// TIA Portal V16 export
// export: Created 2024-09-05T17:39:25.2593397Z, ExportSetting WithDefaults, DisplayName Totally Integrated Automation Portal, DisplayVersion V16 Update 6, DisplayName TIA Portal Version Control Interface, DisplayVersion V16 Update 2, DisplayName TIA Portal Openness, DisplayVersion V16 Update 6, DisplayName STEP 7 Professional, DisplayVersion V16 Update 6, DisplayName STEP 7 Safety, DisplayVersion V16, DisplayName WinCC Advanced, DisplayVersion V16 Update 6
DATA_BLOCK "SET_TIMEZONE_DB"   // DB5
// stored: AutoNumber true, DBAccessibleFromOPCUA true, InstanceOfName SET_TIMEZONE, OfSystemLibElement SET_TIMEZONE, OfSystemLibVersion 2.0
"SET_TIMEZONE"
   // VAR_INPUT
   //    REQ { ExternalAccessible := 'False'; ExternalVisible := 'False'; ExternalWritable := 'False'} : Bool;
   //    TimeZone { ExternalAccessible := 'False'; ExternalVisible := 'False'; ExternalWritable := 'False'} : TimeTransformationRule;
   // END_VAR
   // VAR_OUTPUT
   //    DONE : Bool;
   //    BUSY : Bool;
   //    ERROR : Bool;
   //    STATUS : Word;
   // END_VAR
   // VAR
   //    BusyState : Word;
   //    LastScanREQ { S7_SetPoint := 'True'} : Bool;
   // END_VAR
BEGIN
END_DATA_BLOCK
